// Mitsubishi GX Works2 project: 鹿島外環FLEX   PLC: Q06H
// 鹿島外環ロスゼロ

PROGRAM FLEXPIWI  // PID演算 for WIndows
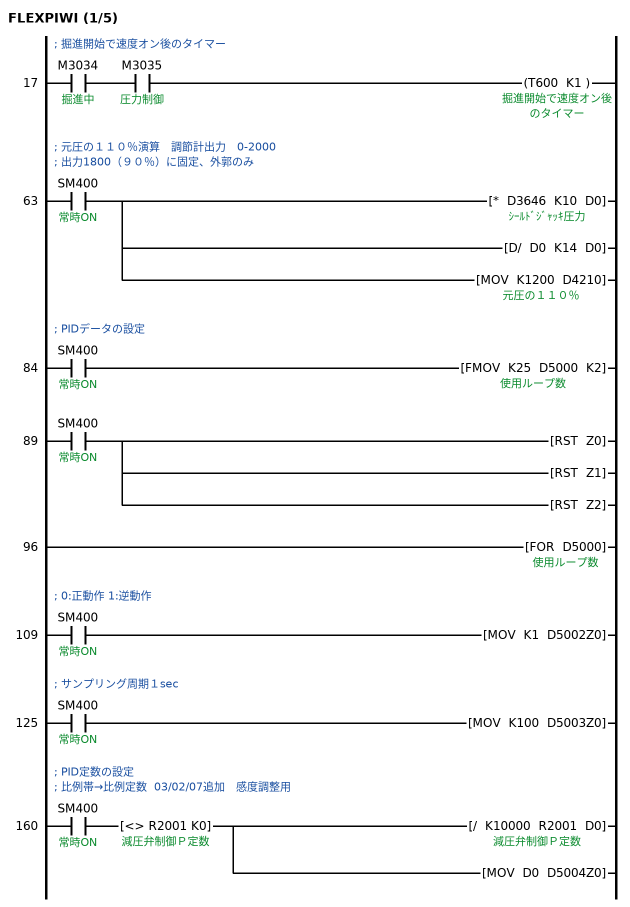
; 掘進開始で速度オン後のタイマー
17    LD      M3034  ; 掘進中
      AND     M3035  ; 圧力制御
      OUT     T600 K1  ; 掘進開始で速度オン後のタイマー
; 元圧の１１０％演算　調節計出力　0-2000
; 出力1800（９０％）に固定、外郭のみ
63    LD      SM400  ; 常時ON
      *       D3646 K10 D0  ; ｼｰﾙﾄﾞｼﾞｬｯｷ圧力
      D/      D0 K14 D0
      MOV     K1200 D4210  ; 元圧の１１０％
; PIDデータの設定
84    LD      SM400  ; 常時ON
      FMOV    K25 D5000 K2  ; 使用ループ数
89    LD      SM400  ; 常時ON
      RST     Z0
      RST     Z1
      RST     Z2
96    FOR     D5000
; 0:正動作 1:逆動作
109   LD      SM400  ; 常時ON
      MOV     K1 D5002Z0
; サンプリング周期１sec
125   LD      SM400  ; 常時ON
      MOV     K100 D5003Z0
; PID定数の設定
; 比例帯→比例定数  03/02/07追加　感度調整用
160   LD      SM400  ; 常時ON
      AND<>   R2001 K0  ; 減圧弁制御Ｐ定数
      /       K10000 R2001 D0
      MOV     D0 D5004Z0
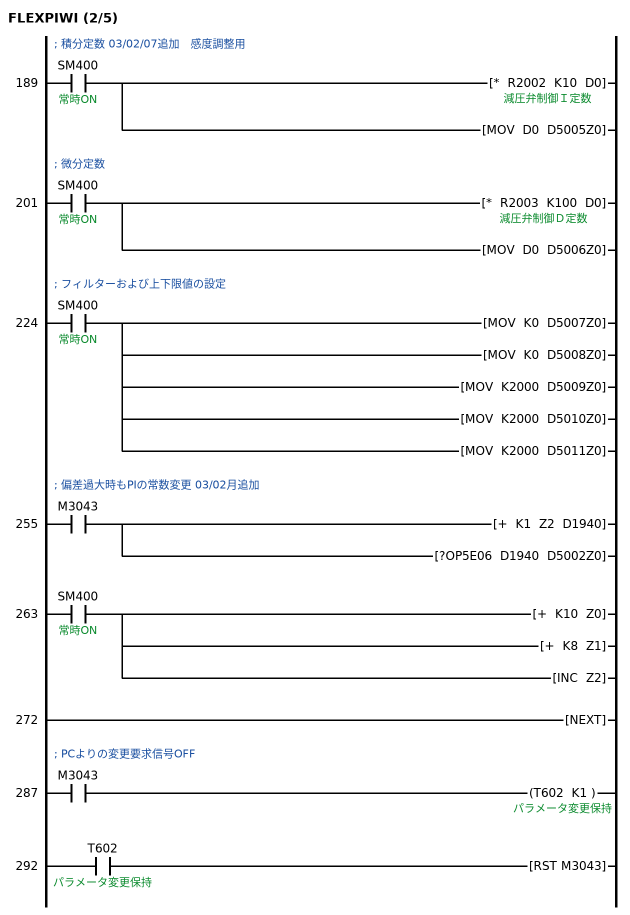
; 積分定数 03/02/07追加　感度調整用
189   LD      SM400  ; 常時ON
      *       R2002 K10 D0  ; 減圧弁制御Ｉ定数
      MOV     D0 D5005Z0
; 微分定数
201   LD      SM400  ; 常時ON
      *       R2003 K100 D0  ; 減圧弁制御Ｄ定数
      MOV     D0 D5006Z0
; フィルターおよび上下限値の設定
224   LD      SM400  ; 常時ON
      MOV     K0 D5007Z0
      MOV     K0 D5008Z0
      MOV     K2000 D5009Z0
      MOV     K2000 D5010Z0
      MOV     K2000 D5011Z0
; 偏差過大時もPIの常数変更 03/02月追加
255   LD      M3043
      +       K1 Z2 D1940
      ?OP5E06 D1940 D5002Z0
263   LD      SM400  ; 常時ON
      +       K10 Z0
      +       K8 Z1
      INC     Z2
272   NEXT
; PCよりの変更要求信号OFF
287   LD      M3043
      OUT     T602 K1  ; パラメータ変更保持
292   LD      T602  ; パラメータ変更保持
      RST     M3043
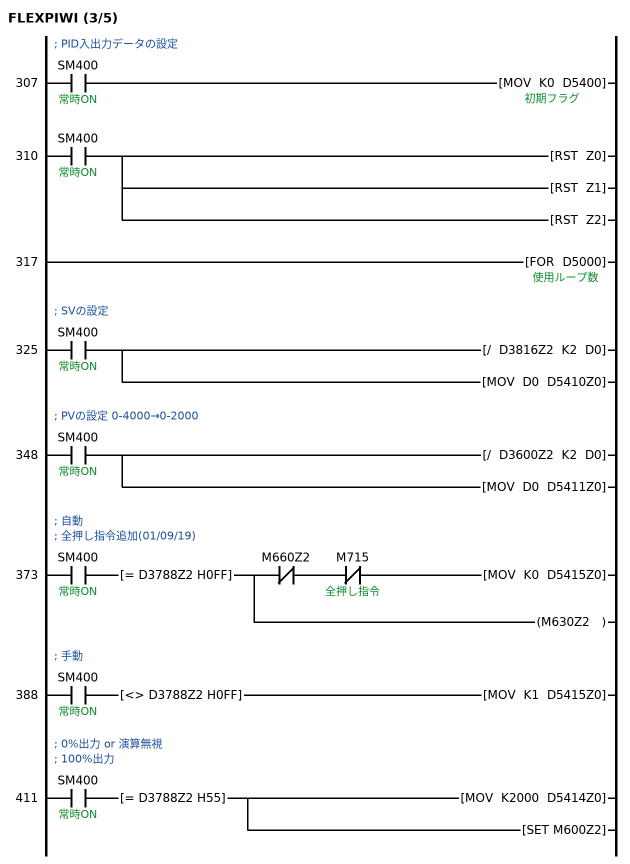
; PID入出力データの設定
307   LD      SM400  ; 常時ON
      MOV     K0 D5400  ; 初期フラグ
310   LD      SM400  ; 常時ON
      RST     Z0
      RST     Z1
      RST     Z2
317   FOR     D5000
; SVの設定
325   LD      SM400  ; 常時ON
      /       D3816Z2 K2 D0
      MOV     D0 D5410Z0
; 
; PVの設定 0-4000→0-2000
348   LD      SM400  ; 常時ON
      /       D3600Z2 K2 D0
      MOV     D0 D5411Z0
; 自動
; 全押し指令追加(01/09/19)
373   LD      SM400  ; 常時ON
      AND=    D3788Z2 H0FF
      MPS
      ANI     M660Z2
      ANI     M715  ; 全押し指令
      MOV     K0 D5415Z0
      MPP
      OUT     M630Z2
; 手動
388   LD      SM400  ; 常時ON
      AND<>   D3788Z2 H0FF
      MOV     K1 D5415Z0
; 0%出力 or 演算無視
; 100%出力
411   LD      SM400  ; 常時ON
      AND=    D3788Z2 H55
      MOV     K2000 D5414Z0
      SET     M600Z2
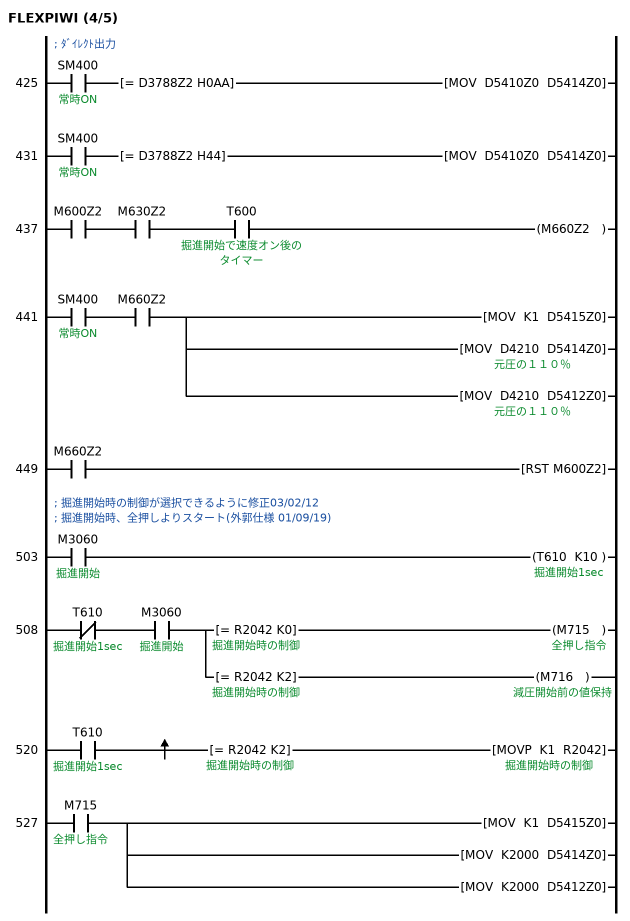
; ﾀﾞｲﾚｸﾄ出力
425   LD      SM400  ; 常時ON
      AND=    D3788Z2 H0AA
      MOV     D5410Z0 D5414Z0
431   LD      SM400  ; 常時ON
      AND=    D3788Z2 H44
      MOV     D5410Z0 D5414Z0
437   LD      M600Z2
      AND     M630Z2
      AND     T600  ; 掘進開始で速度オン後のタイマー
      OUT     M660Z2
441   LD      SM400  ; 常時ON
      AND     M660Z2
      MOV     K1 D5415Z0
      MOV     D4210 D5414Z0
      MOV     D4210 D5412Z0
449   LD      M660Z2
      RST     M600Z2
; 掘進開始時の制御が選択できるように修正03/02/12
; 掘進開始時、全押しよりスタート(外郭仕様 01/09/19)
503   LD      M3060  ; 掘進開始
      OUT     T610 K10  ; 掘進開始1sec
508   LDI     T610  ; 掘進開始1sec
      AND     M3060  ; 掘進開始
      MPS
      AND=    R2042 K0  ; 掘進開始時の制御
      OUT     M715  ; 全押し指令
      MPP
      AND=    R2042 K2  ; 掘進開始時の制御
      OUT     M716  ; 減圧開始前の値保持
520   LD      T610  ; 掘進開始1sec
      MEP
      AND=    R2042 K2  ; 掘進開始時の制御
      MOVP    K1 R2042
527   LD      M715  ; 全押し指令
      MOV     K1 D5415Z0
      MOV     K2000 D5414Z0
      MOV     K2000 D5412Z0
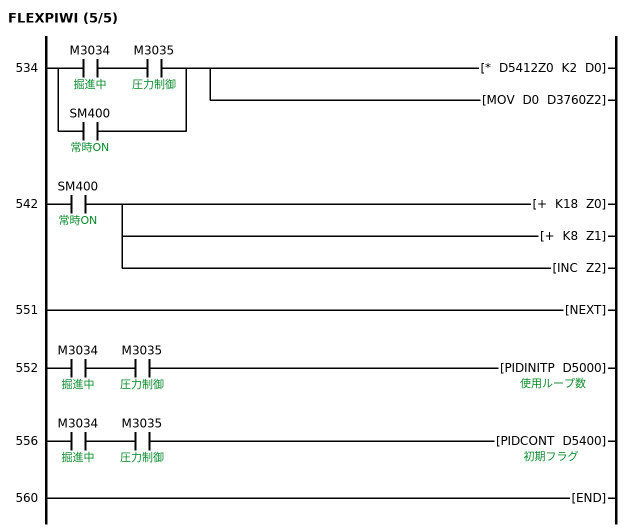
534   LD      M3034  ; 掘進中
      AND     M3035  ; 圧力制御
      OR      SM400  ; 常時ON
      *       D5412Z0 K2 D0
      MOV     D0 D3760Z2
542   LD      SM400  ; 常時ON
      +       K18 Z0
      +       K8 Z1
      INC     Z2
551   NEXT
552   LD      M3034  ; 掘進中
      AND     M3035  ; 圧力制御
      PIDINITP D5000
556   LD      M3034  ; 掘進中
      AND     M3035  ; 圧力制御
      PIDCONT D5400
560   END
END_PROGRAM

PROGRAM FLEXWIN  // FlexWindos対応
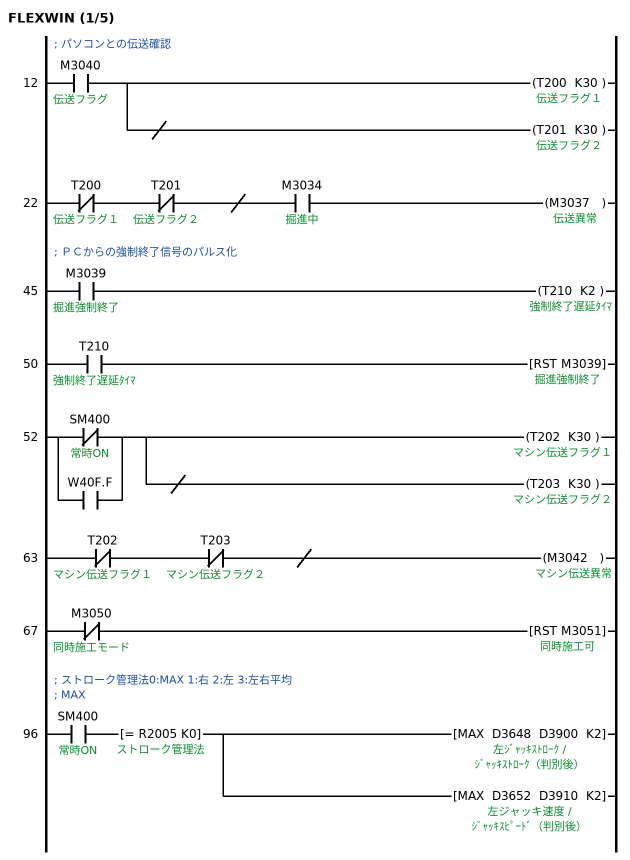
; パソコンとの伝送確認
12    LD      M3040  ; 伝送フラグ
      OUT     T200 K30  ; 伝送フラグ１
      INV
      OUT     T201 K30  ; 伝送フラグ２
22    LDI     T200  ; 伝送フラグ１
      ANI     T201  ; 伝送フラグ２
      INV
      AND     M3034  ; 掘進中
      OUT     M3037  ; 伝送異常
; ＰＣからの強制終了信号のパルス化
45    LD      M3039  ; 掘進強制終了
      OUT     T210 K2  ; 強制終了遅延ﾀｲﾏ
50    LD      T210  ; 強制終了遅延ﾀｲﾏ
      RST     M3039  ; 掘進強制終了
52    LDI     SM400  ; 常時ON
      OR      W40F.F
      OUT     T202 K30  ; マシン伝送フラグ１
      INV
      OUT     T203 K30  ; マシン伝送フラグ２
63    LDI     T202  ; マシン伝送フラグ１
      ANI     T203  ; マシン伝送フラグ２
      INV
      OUT     M3042  ; マシン伝送異常
67    LDI     M3050  ; 同時施工モード
      RST     M3051  ; 同時施工可
; ストローク管理法0:MAX 1:右 2:左 3:左右平均
; MAX
96    LD      SM400  ; 常時ON
      AND=    R2005 K0  ; ストローク管理法
      MAX     D3648 D3900 K2  ; 左ｼﾞｬｯｷｽﾄﾛｰｸ / ｼﾞｬｯｷｽﾄﾛｰｸ（判別後）
      MAX     D3652 D3910 K2  ; 左ジャッキ速度 / ｼﾞｬｯｷｽﾋﾟｰﾄﾞ（判別後）
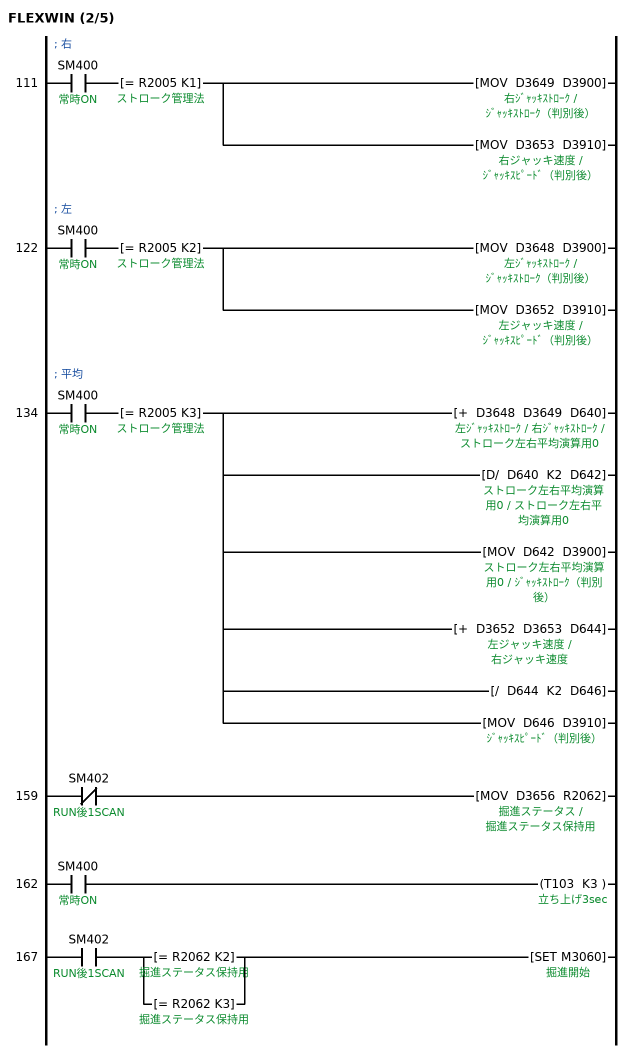
; 右
111   LD      SM400  ; 常時ON
      AND=    R2005 K1  ; ストローク管理法
      MOV     D3649 D3900  ; 右ｼﾞｬｯｷｽﾄﾛｰｸ
      MOV     D3653 D3910  ; 右ジャッキ速度
; 左
122   LD      SM400  ; 常時ON
      AND=    R2005 K2  ; ストローク管理法
      MOV     D3648 D3900
      MOV     D3652 D3910
; 平均
134   LD      SM400  ; 常時ON
      AND=    R2005 K3  ; ストローク管理法
      +       D3648 D3649 D640  ; ストローク左右平均演算用0
      D/      D640 K2 D642  ; ストローク左右平均演算用0
      MOV     D642 D3900
      +       D3652 D3653 D644
      /       D644 K2 D646
      MOV     D646 D3910
159   LDI     SM402  ; RUN後1SCAN
      MOV     D3656 R2062  ; 掘進ステータス / 掘進ステータス保持用
162   LD      SM400  ; 常時ON
      OUT     T103 K3  ; 立ち上げ3sec
167   LD      SM402  ; RUN後1SCAN
      LD=     R2062 K2  ; 掘進ステータス保持用
      OR=     R2062 K3  ; 掘進ステータス保持用
      ANB
      SET     M3060  ; 掘進開始
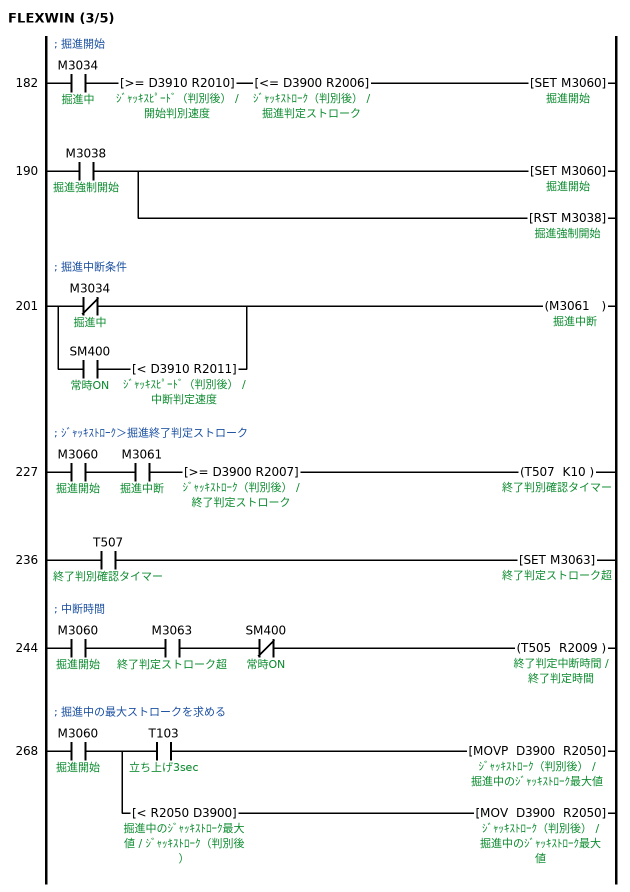
; 掘進開始
182   LD      M3034  ; 掘進中
      AND>=   D3910 R2010  ; ｼﾞｬｯｷｽﾋﾟｰﾄﾞ（判別後） / 開始判別速度
      AND<=   D3900 R2006  ; ｼﾞｬｯｷｽﾄﾛｰｸ（判別後） / 掘進判定ストローク
      SET     M3060  ; 掘進開始
190   LD      M3038  ; 掘進強制開始
      SET     M3060  ; 掘進開始
      RST     M3038  ; 掘進強制開始
; 掘進中断条件
201   LDI     M3034  ; 掘進中
      LD      SM400  ; 常時ON
      AND<    D3910 R2011  ; ｼﾞｬｯｷｽﾋﾟｰﾄﾞ（判別後） / 中断判定速度
      ORB
      OUT     M3061  ; 掘進中断
; ｼﾞｬｯｷｽﾄﾛｰｸ＞掘進終了判定ストローク
227   LD      M3060  ; 掘進開始
      AND     M3061  ; 掘進中断
      AND>=   D3900 R2007  ; ｼﾞｬｯｷｽﾄﾛｰｸ（判別後） / 終了判定ストローク
      OUT     T507 K10  ; 終了判別確認タイマー
236   LD      T507  ; 終了判別確認タイマー
      SET     M3063  ; 終了判定ストローク超
; 中断時間
244   LD      M3060  ; 掘進開始
      AND     M3063  ; 終了判定ストローク超
      ANI     SM400  ; 常時ON
      OUT     T505 R2009  ; 終了判定中断時間 / 終了判定時間
; 掘進中の最大ストロークを求める
268   LD      M3060  ; 掘進開始
      MPS
      AND     T103  ; 立ち上げ3sec
      MOVP    D3900 R2050  ; 掘進中のｼﾞｬｯｷｽﾄﾛｰｸ最大値
      MPP
      AND<    R2050 D3900  ; 掘進中のｼﾞｬｯｷｽﾄﾛｰｸ最大値 / ｼﾞｬｯｷｽﾄﾛｰｸ（判別後）
      MOV     D3900 R2050
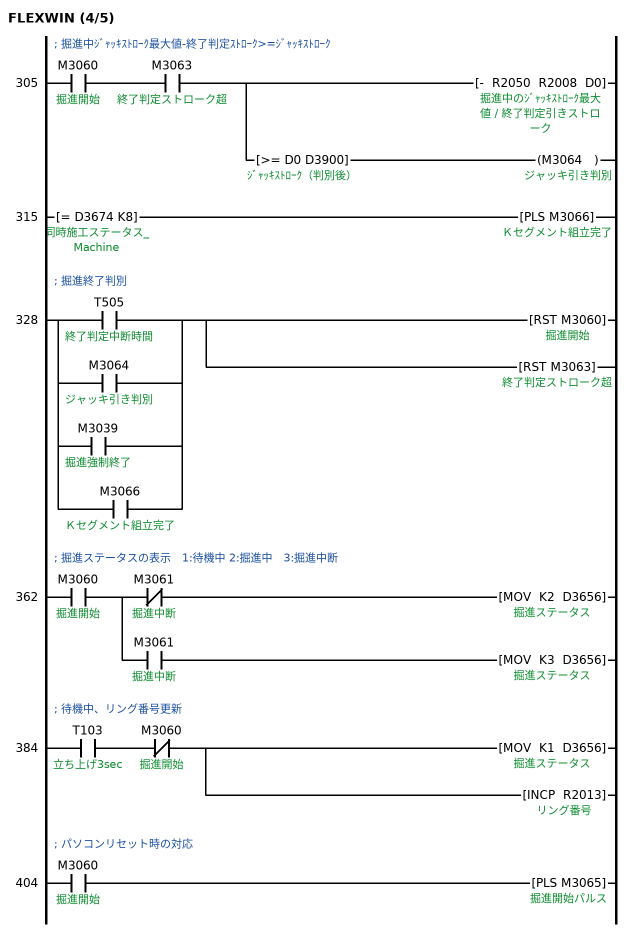
; 掘進中ｼﾞｬｯｷｽﾄﾛｰｸ最大値-終了判定ｽﾄﾛｰｸ>=ｼﾞｬｯｷｽﾄﾛｰｸ
305   LD      M3060  ; 掘進開始
      AND     M3063  ; 終了判定ストローク超
      -       R2050 R2008 D0  ; 終了判定引きストローク
      AND>=   D0 D3900  ; ｼﾞｬｯｷｽﾄﾛｰｸ（判別後）
      OUT     M3064  ; ジャッキ引き判別
315   LD=     D3674 K8  ; 同時施工ステータス_Machine
      PLS     M3066  ; Ｋセグメント組立完了
; 掘進終了判別
328   LD      T505  ; 終了判定中断時間
      OR      M3064  ; ジャッキ引き判別
      OR      M3039  ; 掘進強制終了
      OR      M3066  ; Ｋセグメント組立完了
      RST     M3060  ; 掘進開始
      RST     M3063  ; 終了判定ストローク超
; 掘進ステータスの表示　1:待機中 2:掘進中　3:掘進中断
362   LD      M3060  ; 掘進開始
      MPS
      ANI     M3061  ; 掘進中断
      MOV     K2 D3656
      MPP
      AND     M3061  ; 掘進中断
      MOV     K3 D3656
; 待機中、リング番号更新
384   LD      T103  ; 立ち上げ3sec
      ANI     M3060  ; 掘進開始
      MOV     K1 D3656
      INCP    R2013  ; リング番号
; パソコンリセット時の対応
404   LD      M3060  ; 掘進開始
      PLS     M3065  ; 掘進開始パルス
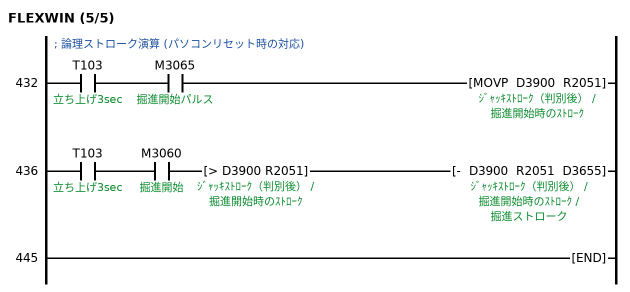
; 論理ストローク演算 (パソコンリセット時の対応)
432   LD      T103  ; 立ち上げ3sec
      AND     M3065  ; 掘進開始パルス
      MOVP    D3900 R2051  ; 掘進開始時のｽﾄﾛｰｸ
436   LD      T103  ; 立ち上げ3sec
      AND     M3060  ; 掘進開始
      AND>    D3900 R2051  ; ｼﾞｬｯｷｽﾄﾛｰｸ（判別後） / 掘進開始時のｽﾄﾛｰｸ
      -       D3900 R2051 D3655  ; 掘進ストローク
445   END
END_PROGRAM

PROGRAM INOUTWIN  // 飛島JS市川
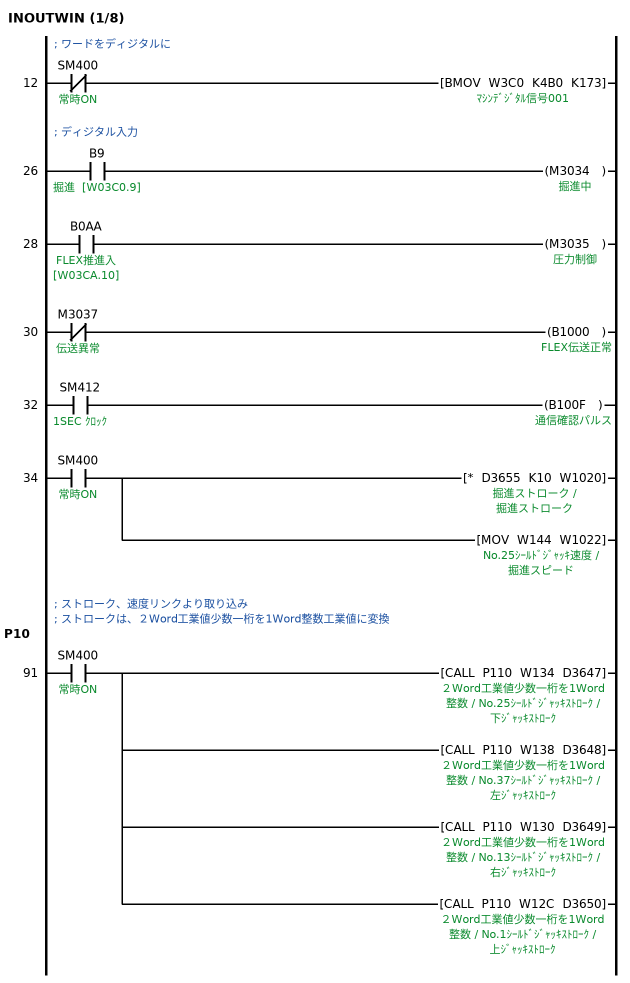
; ワードをディジタルに
12    LDI     SM400  ; 常時ON
      BMOV    W3C0 K4B0 K173  ; ﾏｼﾝﾃﾞｼﾞﾀﾙ信号001 / 中央操作  [W03C0.0]
; ディジタル入力
26    LD      B9  ; 掘進  [W03C0.9]
      OUT     M3034  ; 掘進中
28    LD      B0AA  ; FLEX推進入  [W03CA.10]
      OUT     M3035  ; 圧力制御
30    LDI     M3037  ; 伝送異常
      OUT     B1000  ; FLEX伝送正常
32    LD      SM412  ; 1SEC ｸﾛｯｸ
      OUT     B100F  ; 通信確認パルス
34    LD      SM400  ; 常時ON
      *       D3655 K10 W1020  ; 掘進ストローク / 掘進ストローク
      MOV     W144 W1022  ; No.25ｼｰﾙﾄﾞｼﾞｬｯｷ速度 / 掘進スピード
; ストローク、速度リンクより取り込み
; ストロークは、２Word工業値少数一桁を1Word整数工業値に変換
      P10
91    LD      SM400  ; 常時ON
      CALL    P110 W134 D3647  ; ２Word工業値少数一桁を1Word整数 / No.25ｼｰﾙﾄﾞｼﾞｬｯｷｽﾄﾛｰｸ / 下ｼﾞｬｯｷｽﾄﾛｰｸ
      CALL    P110 W138 D3648  ; No.37ｼｰﾙﾄﾞｼﾞｬｯｷｽﾄﾛｰｸ / 左ｼﾞｬｯｷｽﾄﾛｰｸ
      CALL    P110 W130 D3649  ; No.13ｼｰﾙﾄﾞｼﾞｬｯｷｽﾄﾛｰｸ / 右ｼﾞｬｯｷｽﾄﾛｰｸ
      CALL    P110 W12C D3650  ; No.1ｼｰﾙﾄﾞｼﾞｬｯｷｽﾄﾛｰｸ / 上ｼﾞｬｯｷｽﾄﾛｰｸ
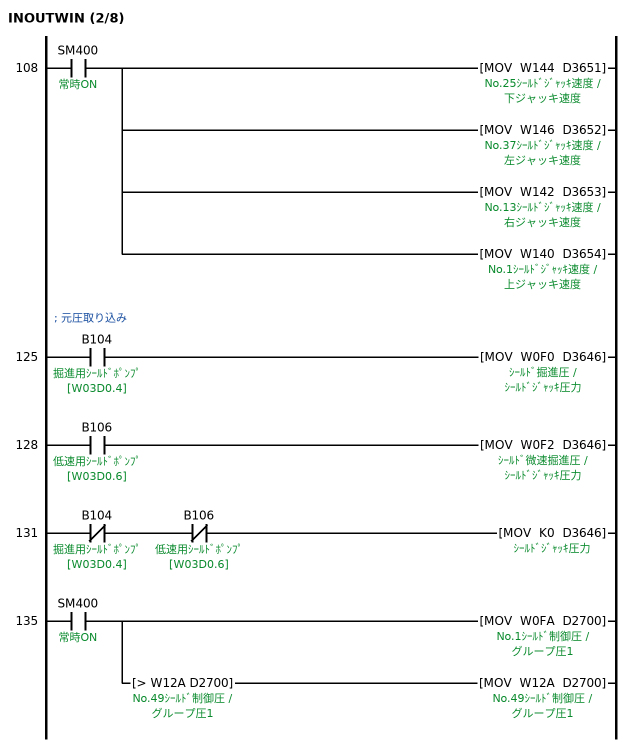
108   LD      SM400  ; 常時ON
      MOV     W144 D3651  ; 下ジャッキ速度
      MOV     W146 D3652  ; No.37ｼｰﾙﾄﾞｼﾞｬｯｷ速度 / 左ジャッキ速度
      MOV     W142 D3653  ; No.13ｼｰﾙﾄﾞｼﾞｬｯｷ速度 / 右ジャッキ速度
      MOV     W140 D3654  ; No.1ｼｰﾙﾄﾞｼﾞｬｯｷ速度 / 上ジャッキ速度
; 元圧取り込み
125   LD      B104  ; 掘進用ｼｰﾙﾄﾞﾎﾟﾝﾌﾟ  [W03D0.4]
      MOV     W0F0 D3646  ; ｼｰﾙﾄﾞ掘進圧 / ｼｰﾙﾄﾞｼﾞｬｯｷ圧力
128   LD      B106  ; 低速用ｼｰﾙﾄﾞﾎﾟﾝﾌﾟ  [W03D0.6]
      MOV     W0F2 D3646  ; ｼｰﾙﾄﾞ微速掘進圧
131   LDI     B104  ; 掘進用ｼｰﾙﾄﾞﾎﾟﾝﾌﾟ  [W03D0.4]
      ANI     B106  ; 低速用ｼｰﾙﾄﾞﾎﾟﾝﾌﾟ  [W03D0.6]
      MOV     K0 D3646
135   LD      SM400  ; 常時ON
      MOV     W0FA D2700  ; No.1ｼｰﾙﾄﾞ制御圧 / グループ圧1
      AND>    W12A D2700  ; No.49ｼｰﾙﾄﾞ制御圧 / グループ圧1
      MOV     W12A D2700
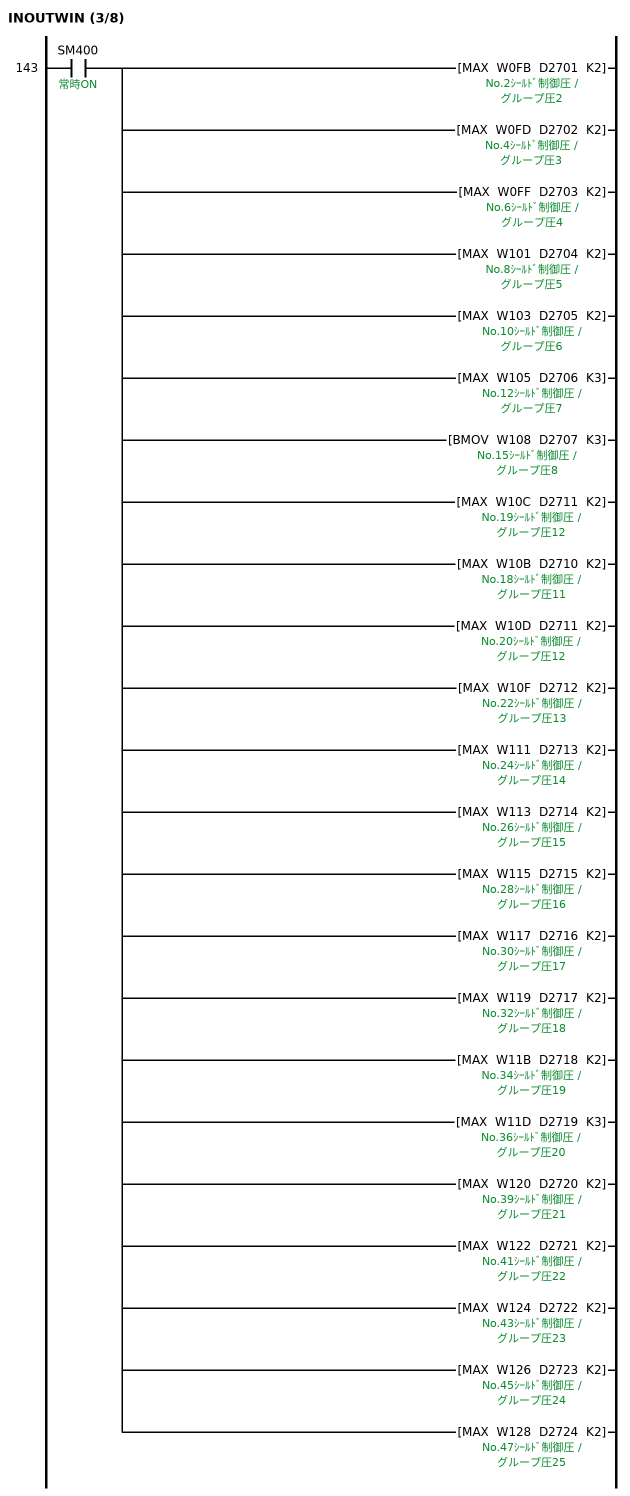
143   LD      SM400  ; 常時ON
      MAX     W0FB D2701 K2  ; No.2ｼｰﾙﾄﾞ制御圧 / グループ圧2
      MAX     W0FD D2702 K2  ; No.4ｼｰﾙﾄﾞ制御圧 / グループ圧3
      MAX     W0FF D2703 K2  ; No.6ｼｰﾙﾄﾞ制御圧 / グループ圧4
      MAX     W101 D2704 K2  ; No.8ｼｰﾙﾄﾞ制御圧 / グループ圧5
      MAX     W103 D2705 K2  ; No.10ｼｰﾙﾄﾞ制御圧 / グループ圧6
      MAX     W105 D2706 K3  ; No.12ｼｰﾙﾄﾞ制御圧 / グループ圧7
      BMOV    W108 D2707 K3  ; No.15ｼｰﾙﾄﾞ制御圧 / グループ圧8
      MAX     W10C D2711 K2  ; No.19ｼｰﾙﾄﾞ制御圧 / グループ圧12
      MAX     W10B D2710 K2  ; No.18ｼｰﾙﾄﾞ制御圧 / グループ圧11
      MAX     W10D D2711 K2  ; No.20ｼｰﾙﾄﾞ制御圧
      MAX     W10F D2712 K2  ; No.22ｼｰﾙﾄﾞ制御圧 / グループ圧13
      MAX     W111 D2713 K2  ; No.24ｼｰﾙﾄﾞ制御圧 / グループ圧14
      MAX     W113 D2714 K2  ; No.26ｼｰﾙﾄﾞ制御圧 / グループ圧15
      MAX     W115 D2715 K2  ; No.28ｼｰﾙﾄﾞ制御圧 / グループ圧16
      MAX     W117 D2716 K2  ; No.30ｼｰﾙﾄﾞ制御圧 / グループ圧17
      MAX     W119 D2717 K2  ; No.32ｼｰﾙﾄﾞ制御圧 / グループ圧18
      MAX     W11B D2718 K2  ; No.34ｼｰﾙﾄﾞ制御圧 / グループ圧19
      MAX     W11D D2719 K3  ; No.36ｼｰﾙﾄﾞ制御圧 / グループ圧20
      MAX     W120 D2720 K2  ; No.39ｼｰﾙﾄﾞ制御圧 / グループ圧21
      MAX     W122 D2721 K2  ; No.41ｼｰﾙﾄﾞ制御圧 / グループ圧22
      MAX     W124 D2722 K2  ; No.43ｼｰﾙﾄﾞ制御圧 / グループ圧23
      MAX     W126 D2723 K2  ; No.45ｼｰﾙﾄﾞ制御圧 / グループ圧24
      MAX     W128 D2724 K2  ; No.47ｼｰﾙﾄﾞ制御圧 / グループ圧25
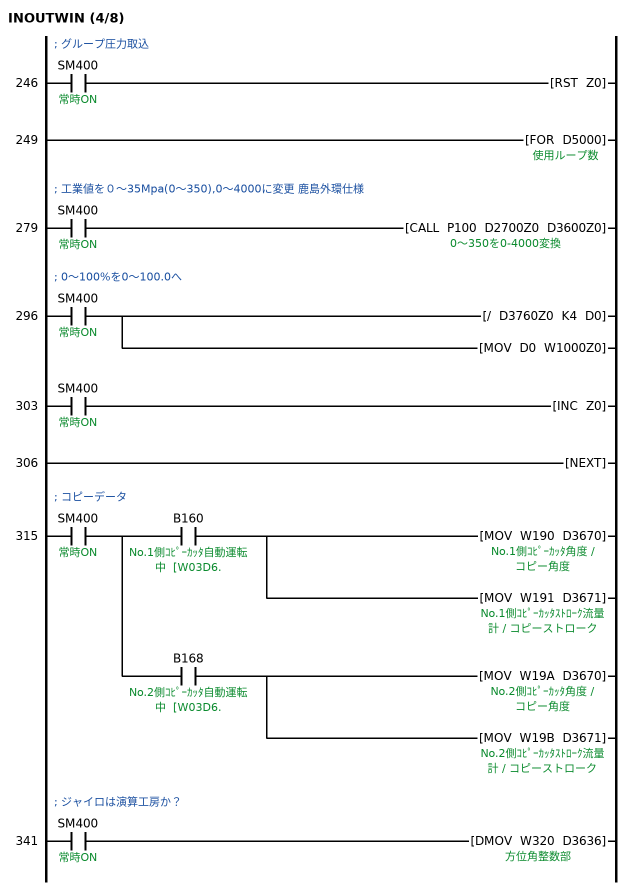
; グループ圧力取込
246   LD      SM400  ; 常時ON
      RST     Z0
249   FOR     D5000  ; 使用ループ数
; 工業値を０～35Mpa(0～350),0～4000に変更 鹿島外環仕様
279   LD      SM400  ; 常時ON
      CALL    P100 D2700Z0 D3600Z0  ; 0～350を0-4000変換
; 0～100%を0～100.0へ
296   LD      SM400  ; 常時ON
      /       D3760Z0 K4 D0
      MOV     D0 W1000Z0
303   LD      SM400  ; 常時ON
      INC     Z0
306   NEXT
; コピーデータ
315   LD      SM400  ; 常時ON
      MPS
      AND     B160  ; No.1側ｺﾋﾟｰｶｯﾀ自動運転中  [W03D6.
      MOV     W190 D3670  ; No.1側ｺﾋﾟｰｶｯﾀ角度 / コピー角度
      MOV     W191 D3671  ; No.1側ｺﾋﾟｰｶｯﾀｽﾄﾛｰｸ流量計 / コピーストローク
      MPP
      AND     B168  ; No.2側ｺﾋﾟｰｶｯﾀ自動運転中  [W03D6.
      MOV     W19A D3670  ; No.2側ｺﾋﾟｰｶｯﾀ角度
      MOV     W19B D3671  ; No.2側ｺﾋﾟｰｶｯﾀｽﾄﾛｰｸ流量計
; ジャイロは演算工房か？
341   LD      SM400  ; 常時ON
      DMOV    W320 D3636  ; 方位角整数部
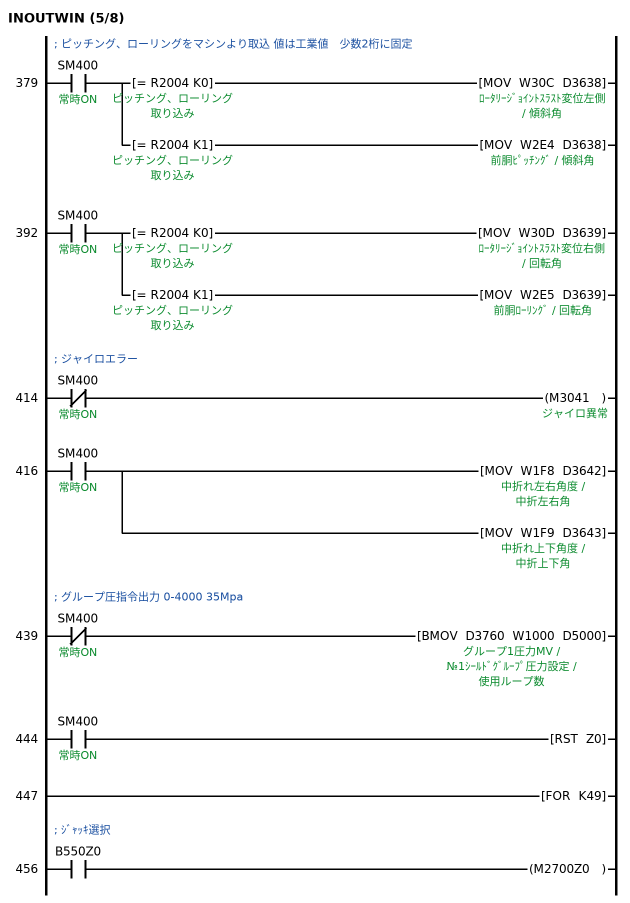
; ピッチング、ローリングをマシンより取込 値は工業値　少数2桁に固定
379   LD      SM400  ; 常時ON
      MPS
      AND=    R2004 K0  ; ピッチング、ローリング取り込み
      MOV     W30C D3638  ; ﾛｰﾀﾘｰｼﾞｮｲﾝﾄｽﾗｽﾄ変位左側 / 傾斜角
      MPP
      AND=    R2004 K1  ; ピッチング、ローリング取り込み
      MOV     W2E4 D3638  ; 前胴ﾋﾟｯﾁﾝｸﾞ
392   LD      SM400  ; 常時ON
      MPS
      AND=    R2004 K0  ; ピッチング、ローリング取り込み
      MOV     W30D D3639  ; ﾛｰﾀﾘｰｼﾞｮｲﾝﾄｽﾗｽﾄ変位右側 / 回転角
      MPP
      AND=    R2004 K1  ; ピッチング、ローリング取り込み
      MOV     W2E5 D3639  ; 前胴ﾛｰﾘﾝｸﾞ
; ジャイロエラー
414   LDI     SM400  ; 常時ON
      OUT     M3041  ; ジャイロ異常
416   LD      SM400  ; 常時ON
      MOV     W1F8 D3642  ; 中折れ左右角度 / 中折左右角
      MOV     W1F9 D3643  ; 中折れ上下角度 / 中折上下角
; グループ圧指令出力 0-4000 35Mpa
439   LDI     SM400  ; 常時ON
      BMOV    D3760 W1000 D5000  ; グループ1圧力MV / №1ｼｰﾙﾄﾞｸﾞﾙｰﾌﾟ圧力設定
444   LD      SM400  ; 常時ON
      RST     Z0
447   FOR     K49
; ｼﾞｬｯｷ選択
456   LD      B550Z0
      OUT     M2700Z0
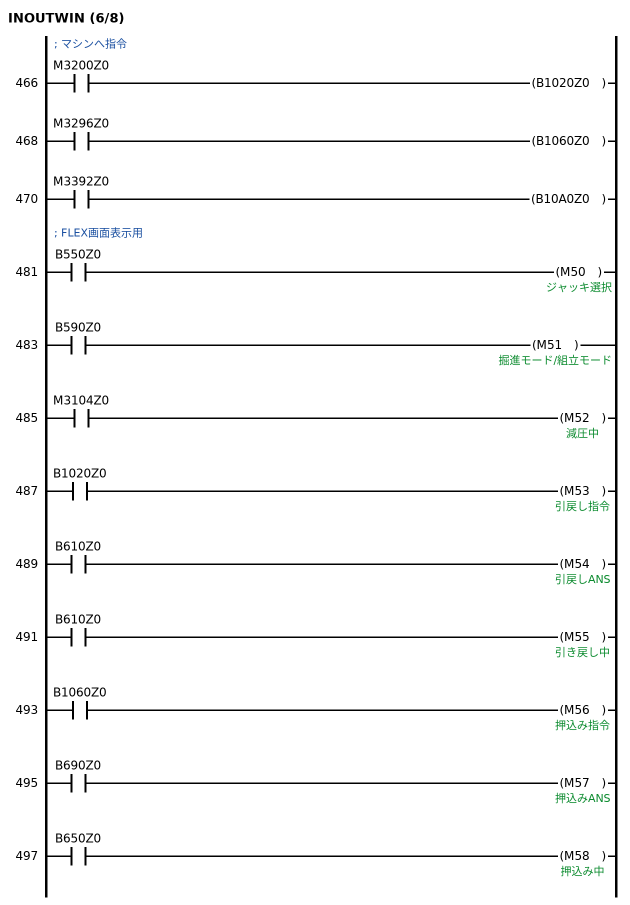
; マシンへ指令
466   LD      M3200Z0
      OUT     B1020Z0
468   LD      M3296Z0
      OUT     B1060Z0
470   LD      M3392Z0
      OUT     B10A0Z0
; FLEX画面表示用
481   LD      B550Z0
      OUT     M50  ; ジャッキ選択
483   LD      B590Z0
      OUT     M51  ; 掘進モード/組立モード
485   LD      M3104Z0
      OUT     M52  ; 減圧中
487   LD      B1020Z0
      OUT     M53  ; 引戻し指令
489   LD      B610Z0
      OUT     M54  ; 引戻しANS
491   LD      B610Z0
      OUT     M55  ; 引き戻し中
493   LD      B1060Z0
      OUT     M56  ; 押込み指令
495   LD      B690Z0
      OUT     M57  ; 押込みANS
497   LD      B650Z0
      OUT     M58  ; 押込み中
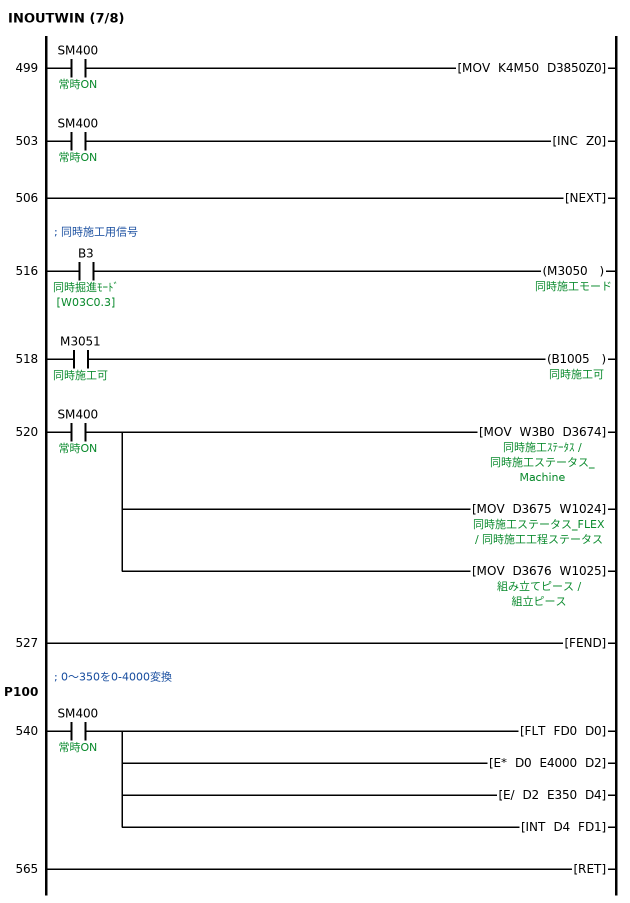
499   LD      SM400  ; 常時ON
      MOV     K4M50 D3850Z0
503   LD      SM400  ; 常時ON
      INC     Z0
506   NEXT
; 同時施工用信号
516   LD      B3  ; 同時掘進ﾓｰﾄﾞ  [W03C0.3]
      OUT     M3050  ; 同時施工モード
518   LD      M3051  ; 同時施工可
      OUT     B1005  ; 同時施工可
520   LD      SM400  ; 常時ON
      MOV     W3B0 D3674  ; 同時施工ｽﾃｰﾀｽ / 同時施工ステータス_Machine
      MOV     D3675 W1024  ; 同時施工ステータス_FLEX / 同時施工工程ステータス
      MOV     D3676 W1025  ; 組み立てピース / 組立ピース
527   FEND
      P100
; 0～350を0-4000変換
540   LD      SM400  ; 常時ON
      FLT     FD0 D0
        [note] スケール上限
      E*      D0 E4000 D2
      E/      D2 E350 D4
      INT     D4 FD1
565   RET
      P110
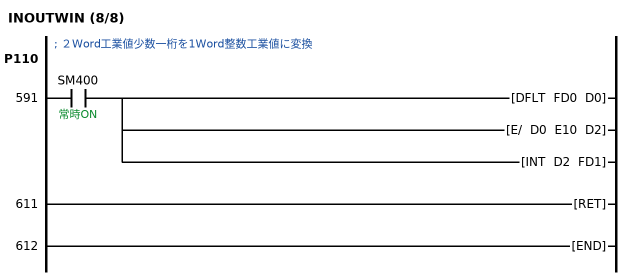
; ２Word工業値少数一桁を1Word整数工業値に変換
591   LD      SM400  ; 常時ON
      DFLT    FD0 D0
        [note] スケール上限
      E/      D0 E10 D2
      INT     D2 FD1
611   RET
612   END
END_PROGRAM

PROGRAM Simlat  // 鹿島外環FLEX
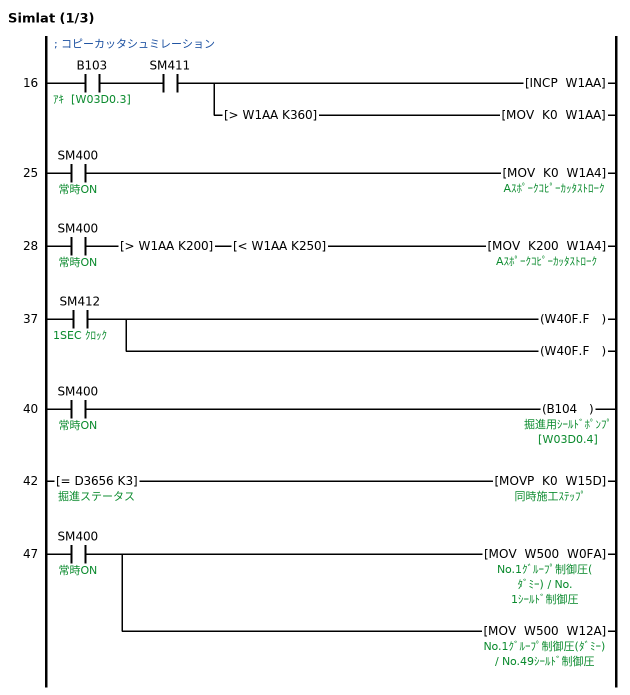
; コピーカッタシュミレーション
16    LD      B103  ; ｱｷ  [W03D0.3]
      AND     SM411
      INCP    W1AA
      AND>    W1AA K360
      MOV     K0 W1AA
25    LD      SM400  ; 常時ON
      MOV     K0 W1A4  ; Aｽﾎﾟｰｸｺﾋﾟｰｶｯﾀｽﾄﾛｰｸ
28    LD      SM400  ; 常時ON
      AND>    W1AA K200
      AND<    W1AA K250
      MOV     K200 W1A4
37    LD      SM412  ; 1SEC ｸﾛｯｸ
      OUT     W40F.F
      OUT     W40F.F
40    LD      SM400  ; 常時ON
      OUT     B104  ; 掘進用ｼｰﾙﾄﾞﾎﾟﾝﾌﾟ  [W03D0.4]
42    LD=     D3656 K3  ; 掘進ステータス
      MOVP    K0 W15D  ; 同時施工ｽﾃｯﾌﾟ
47    LD      SM400  ; 常時ON
      MOV     W500 W0FA  ; No.1ｸﾞﾙｰﾌﾟ制御圧(ﾀﾞﾐｰ) / No.1ｼｰﾙﾄﾞ制御圧
      MOV     W500 W12A  ; No.49ｼｰﾙﾄﾞ制御圧
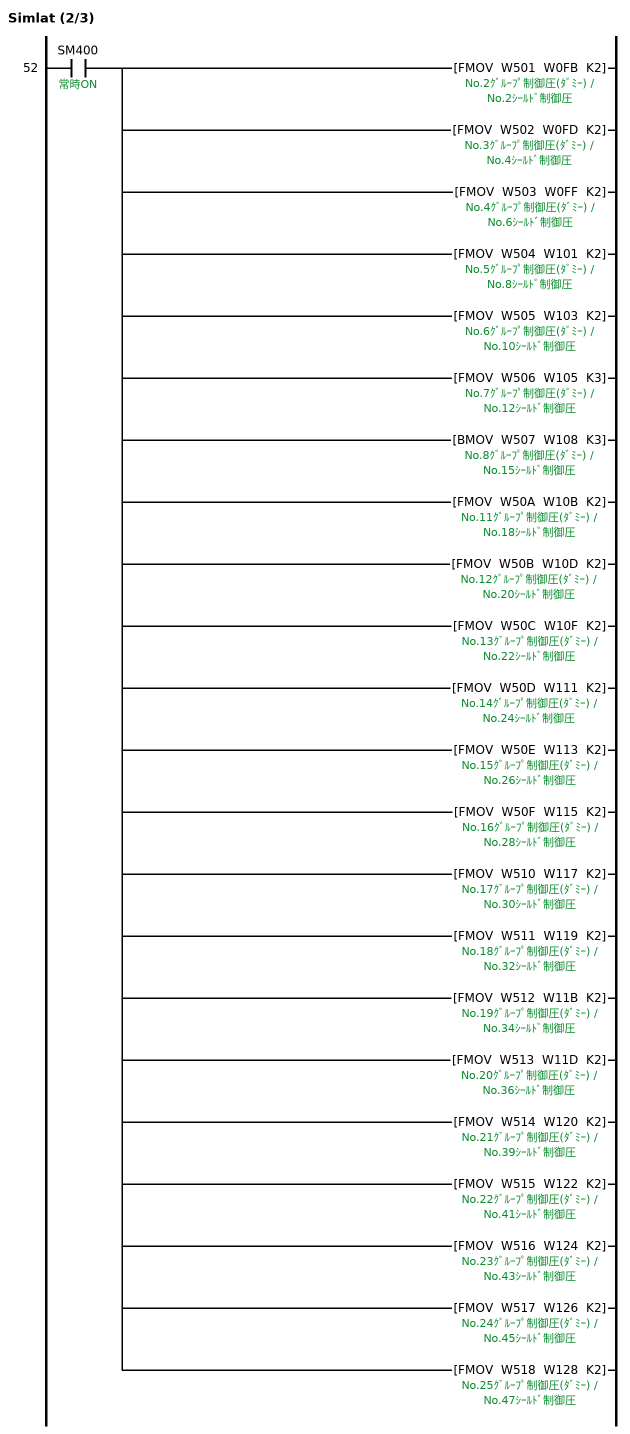
52    LD      SM400  ; 常時ON
      FMOV    W501 W0FB K2  ; No.2ｸﾞﾙｰﾌﾟ制御圧(ﾀﾞﾐｰ) / No.2ｼｰﾙﾄﾞ制御圧
      FMOV    W502 W0FD K2  ; No.3ｸﾞﾙｰﾌﾟ制御圧(ﾀﾞﾐｰ) / No.4ｼｰﾙﾄﾞ制御圧
      FMOV    W503 W0FF K2  ; No.4ｸﾞﾙｰﾌﾟ制御圧(ﾀﾞﾐｰ) / No.6ｼｰﾙﾄﾞ制御圧
      FMOV    W504 W101 K2  ; No.5ｸﾞﾙｰﾌﾟ制御圧(ﾀﾞﾐｰ) / No.8ｼｰﾙﾄﾞ制御圧
      FMOV    W505 W103 K2  ; No.6ｸﾞﾙｰﾌﾟ制御圧(ﾀﾞﾐｰ) / No.10ｼｰﾙﾄﾞ制御圧
      FMOV    W506 W105 K3  ; No.7ｸﾞﾙｰﾌﾟ制御圧(ﾀﾞﾐｰ) / No.12ｼｰﾙﾄﾞ制御圧
      BMOV    W507 W108 K3  ; No.8ｸﾞﾙｰﾌﾟ制御圧(ﾀﾞﾐｰ) / No.15ｼｰﾙﾄﾞ制御圧
      FMOV    W50A W10B K2  ; No.11ｸﾞﾙｰﾌﾟ制御圧(ﾀﾞﾐｰ) / No.18ｼｰﾙﾄﾞ制御圧
      FMOV    W50B W10D K2  ; No.12ｸﾞﾙｰﾌﾟ制御圧(ﾀﾞﾐｰ) / No.20ｼｰﾙﾄﾞ制御圧
      FMOV    W50C W10F K2  ; No.13ｸﾞﾙｰﾌﾟ制御圧(ﾀﾞﾐｰ) / No.22ｼｰﾙﾄﾞ制御圧
      FMOV    W50D W111 K2  ; No.14ｸﾞﾙｰﾌﾟ制御圧(ﾀﾞﾐｰ) / No.24ｼｰﾙﾄﾞ制御圧
      FMOV    W50E W113 K2  ; No.15ｸﾞﾙｰﾌﾟ制御圧(ﾀﾞﾐｰ) / No.26ｼｰﾙﾄﾞ制御圧
      FMOV    W50F W115 K2  ; No.16ｸﾞﾙｰﾌﾟ制御圧(ﾀﾞﾐｰ) / No.28ｼｰﾙﾄﾞ制御圧
      FMOV    W510 W117 K2  ; No.17ｸﾞﾙｰﾌﾟ制御圧(ﾀﾞﾐｰ) / No.30ｼｰﾙﾄﾞ制御圧
      FMOV    W511 W119 K2  ; No.18ｸﾞﾙｰﾌﾟ制御圧(ﾀﾞﾐｰ) / No.32ｼｰﾙﾄﾞ制御圧
      FMOV    W512 W11B K2  ; No.19ｸﾞﾙｰﾌﾟ制御圧(ﾀﾞﾐｰ) / No.34ｼｰﾙﾄﾞ制御圧
      FMOV    W513 W11D K2  ; No.20ｸﾞﾙｰﾌﾟ制御圧(ﾀﾞﾐｰ) / No.36ｼｰﾙﾄﾞ制御圧
      FMOV    W514 W120 K2  ; No.21ｸﾞﾙｰﾌﾟ制御圧(ﾀﾞﾐｰ) / No.39ｼｰﾙﾄﾞ制御圧
      FMOV    W515 W122 K2  ; No.22ｸﾞﾙｰﾌﾟ制御圧(ﾀﾞﾐｰ) / No.41ｼｰﾙﾄﾞ制御圧
      FMOV    W516 W124 K2  ; No.23ｸﾞﾙｰﾌﾟ制御圧(ﾀﾞﾐｰ) / No.43ｼｰﾙﾄﾞ制御圧
      FMOV    W517 W126 K2  ; No.24ｸﾞﾙｰﾌﾟ制御圧(ﾀﾞﾐｰ) / No.45ｼｰﾙﾄﾞ制御圧
      FMOV    W518 W128 K2  ; No.25ｸﾞﾙｰﾌﾟ制御圧(ﾀﾞﾐｰ) / No.47ｼｰﾙﾄﾞ制御圧
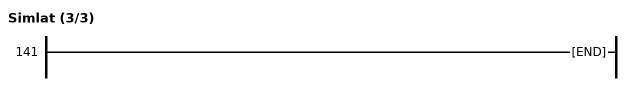
141   END
END_PROGRAM

// device comments not shown above
D3600  ; グループ1圧力
D3816  ; グループ1圧力SV
D5002  ; グループ1演算式選択
D5412  ; グループ1自動操作量（MV)
